Fanuc KAREL source: IO0038.KL

-- PROVISIONAL review KL for V770-1; original PC SHA256 0dc276f8c4e53b844ab1ec3b79d2b44d53d826c4f3ec6fb75ef65a723acfbd69
-- Incomplete behavior may be omitted. Consult companion uncertainty JSON. Do not deploy.
PROGRAM IO0038
%NOLOCKGROUP
-- UNRESOLVED_LOCAL_POOL 5 cells at code offset 13; source declarations unknown
-- DIRECT_LOCAL_WORD_ACCESS alone does not prove INTEGER, REAL, or BOOLEAN
BEGIN
  -- UNRESOLVED_PC offsets 0-18; opcodes 2B,2C,7B
  -- UNRESOLVED_PC offsets 23-30; opcodes 9D,23
  -- UNRESOLVED_PC offsets 35-49; opcodes 2E,22,9D,33,35
  -- UNRESOLVED_PC offsets 54-61; opcodes 9D,23
  -- UNRESOLVED_PC offsets 66-77; opcodes 2E,23
  -- UNRESOLVED_PC offsets 82-95; opcodes 2E,19,23
  -- UNRESOLVED_PC offsets 100-104; opcodes 7F
  -- UNRESOLVED_PC offsets 109-113; opcodes 27,AA
  -- UNRESOLVED_PC offsets 118-122; opcodes 7F
END IO0038
